{attribute addProperty BoxType "KL6821"}
{attribute addProperty Id "Channel_1Channel_0A9F16DB00"}
{attribute addProperty CRC "839001755"}
{attribute addProperty SizeInBites "0"}
{attribute addProperty SizeInBytes "0"}
TYPE KL6821_3202269B :
STRUCT
	{attribute addProperty Name "Channel_1"}
	Channel_1 : Channel_0A9F16DB;
END_STRUCT
END_TYPE

(* stored: Version 1.2.0.0, ProductVersion 3.1.4024.9
   DUT KL6821_3202269B: Id {f96ffe38-633d-4870-9f58-d194f486a225} *)
